// TIA Portal project "Control PLC con HMI" (V15.1)

(* hardware
DEVICE "S7-1200 station_1"  S7-1200 Station
   slot 0: "Rack_0"  S7-1200 Rack  Rack  V1.0
   slot 1: "PLC_1"  CPU 1212C AC/DC/Rly  6ES7 212-1BD30-0XB0  V2.2
DEVICE "HMI_1"  KTP400 Basic PN
   slot 0: "KTP400 Basic PN"  KTP400 Basic PN  6AV2 123-2DB03-0AX0  14.0.0.0
   slot 1: "HMI_RT_1"  KTP400 Basic PN  6AV2 123-2DB03-0AX0  14.0.0.0
   slot 5: "HMI_1.IE_CP_1"  PROFINET Interface  14.0.0.0
      slot 1: "Interfaz PROFINET_1"  PROFINET Interface
         slot 1: "Port_1"  Port
*)

// ===== PLC "PLC_1"  CPU 1212C AC/DC/Rly =====

VAR_GLOBAL   // PLC tag table "Tabla de variables estándar"
   "Q contador" AT %M0.5 : Bool;
   "CV contador" AT %MW20 : Int;
   "PV contador" AT %MW22 : Int;
   "In contador" AT %M24.1 : Bool;
   "Down contador" AT %M0.6 : Bool;
   "QD contador" AT %M1.0 : Bool;
   "Reset contador semaforo" AT %M1.1 : Bool;
   "CV contador semaforo" AT %MW30 : Int;
   "semaforo rojo" AT %M1.2 : Bool;
   "semaforo naranja" AT %M1.3 : Bool;
   "semaforo verde" AT %M1.4 : Bool;
   "Tempo" AT %M1.5 : Bool;
   "Entrada analogica 1" AT %IW66 : Int;
   "Senal escalada 1" AT %MD32 : Real;
   "Alarma up" AT %M1.6 : Bool;
   "Alarma down" AT %M1.7 : Bool;
END_VAR

VAR_GLOBAL   // PLC tag table "Entradas"
   "ARRANQUE" AT %I0.0 : Bool;
   "PARO" AT %I0.1 : Bool;
   "Senal analogica 0" AT %IW64 : Int;
END_VAR

VAR_GLOBAL   // PLC tag table "Salidas"
   "MOTOR1" AT %Q0.0 : Bool;
END_VAR

VAR_GLOBAL   // PLC tag table "Memoria"
   "Senal analogica real 0" AT %MD2 : Real;
   "Segundos" AT %MD26 : Time;
   "senal escalada" AT %MD6 : Real;
   "Senal de control" AT %M0.2 : Bool;
END_VAR

VAR_GLOBAL   // PLC tag table "HMI"
   "ARRANQUE HMI" AT %M0.0 : Bool;
   "PARO HMI" AT %M0.1 : Bool;
   "Reset contador" AT %M24.0 : Bool;
   "Q timer" AT %M0.3 : Bool;
   "Et timer" AT %MD10 : Time;
   "Pt Timer" AT %MD14 : Time;
   "in timer" AT %M18.0 : Bool;
   "Reset timer" AT %M0.4 : Bool;
   "Load contador" AT %M0.7 : Bool;
END_VAR

DATA_BLOCK "Control analogico_DB"   // DB5
{ S7_Optimized_Access := 'TRUE' }
VERSION : 0.1
// stored: InstanceOfName Control analogico
"Control analogico"
BEGIN
END_DATA_BLOCK

// folder: System blocks/Program resources

DATA_BLOCK "IEC_Timer_0_DB"   // DB1
{ S7_Optimized_Access := 'TRUE' }
AUTHOR : Simatic
FAMILY : IEC
NAME : IEC_TMR
VERSION : 1.0
// stored: InstanceOfName IEC_TIMER
"IEC_TIMER"
BEGIN
END_DATA_BLOCK

DATA_BLOCK "IEC_Counter_0_DB"   // DB2
{ S7_Optimized_Access := 'TRUE' }
AUTHOR : Simatic
FAMILY : IEC
NAME : CNTR
VERSION : 1.0
// stored: InstanceOfName IEC_COUNTER
"IEC_COUNTER"
BEGIN
END_DATA_BLOCK

DATA_BLOCK "IEC_Timer_0_DB_1"   // DB3
{ S7_Optimized_Access := 'TRUE' }
AUTHOR : Simatic
FAMILY : IEC
NAME : IEC_TMR
VERSION : 1.0
// stored: InstanceOfName IEC_TIMER
"IEC_TIMER"
BEGIN
END_DATA_BLOCK

DATA_BLOCK "IEC_Counter_0_DB_1"   // DB4
{ S7_Optimized_Access := 'TRUE' }
AUTHOR : Simatic
FAMILY : IEC
NAME : CNTR
VERSION : 1.0
// stored: InstanceOfName IEC_COUNTER
"IEC_COUNTER"
BEGIN
END_DATA_BLOCK

// folder: (top level)

FUNCTION_BLOCK "Control analogico"   // FB1, LAD
{ S7_Optimized_Access := 'TRUE' }
VERSION : 0.1
   VAR_INPUT
      "Entrada analogica" : DInt;
      Minimo : Real;
      Maximo : Real;
      "Alarm max" : Real;
      "Alarm min" : Real;
   END_VAR
   VAR_OUTPUT
      "Senal out" : Real;
      "Alarm up" : Bool;
      "Alarm down" : Bool;
   END_VAR
   VAR_TEMP
      "Sinal norm" : Real;
   END_VAR
BEGIN

REGION Network 1
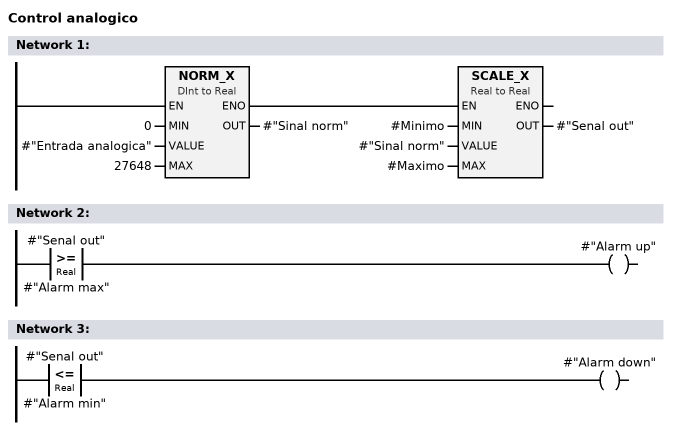
   RUNG wire#powerrail
      { S7_Templates := "[SrcType := DInt, DestType := Real]"; S7_GenerateENO := "TRUE" } Normalize(min := 0, value := #"Entrada analogica", max := 27648, out => #"Sinal norm")
      { S7_Templates := "[SrcType := Real, DestType := Real]"; S7_GenerateENO := "TRUE" } Scale(min := #Minimo, value := #"Sinal norm", max := #Maximo, out => #"Senal out")
   END_RUNG
   // the same network as SCL:
   // ENO of a box is taken as its EN; it also drops when the box reports an error
   #"Sinal norm" := NORM_X(MIN := 0, VALUE := #"Entrada analogica", MAX := 27648);
   #"Senal out" := SCALE_X(MIN := #Minimo, VALUE := #"Sinal norm", MAX := #Maximo);
END_REGION

REGION Network 2
   RUNG wire#powerrail
      { S7_Templates := "SrcType := Real" } GE_Contact(in1 := #"Senal out", in2 := #"Alarm max")
      Coil( #"Alarm up" )
   END_RUNG
   // the same network as SCL:
   #"Alarm up" := #"Senal out" >= #"Alarm max";
END_REGION

REGION Network 3
   RUNG wire#powerrail
      { S7_Templates := "SrcType := Real" } LE_Contact(in1 := #"Senal out", in2 := #"Alarm min")
      Coil( #"Alarm down" )
   END_RUNG
   // the same network as SCL:
   #"Alarm down" := #"Senal out" <= #"Alarm min";
END_REGION
END_FUNCTION_BLOCK

FUNCTION "MOTOR" : Void   // FC1, LAD
{ S7_Optimized_Access := 'TRUE' }
VERSION : 0.1
BEGIN

REGION Network 1
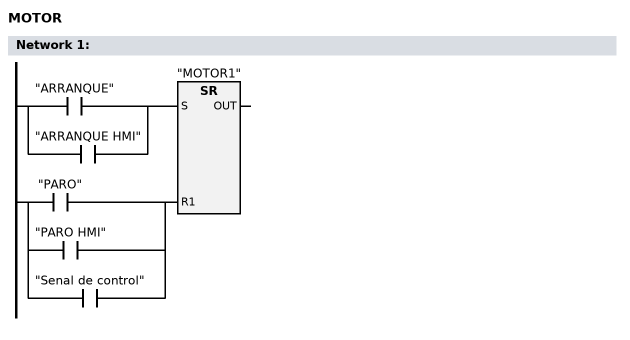
   RUNG wire#powerrail
      Contact( "ARRANQUE" )
      wire#w1
      S_SR(operand := "MOTOR1", r1 := wire#w2)
   END_RUNG
   RUNG wire#powerrail
      Contact( "ARRANQUE HMI" )
   END_RUNG wire#w1
   RUNG wire#powerrail
      Contact( "PARO" )
   END_RUNG wire#w2
   RUNG wire#powerrail
      Contact( "PARO HMI" )
   END_RUNG wire#w2
   RUNG wire#powerrail
      Contact( "Senal de control" )
   END_RUNG wire#w2
   // the same network as SCL:
   IF "ARRANQUE" OR "ARRANQUE HMI" THEN
       "MOTOR1" := TRUE;   // SR flip-flop
   END_IF;
   IF "PARO" OR "PARO HMI" OR "Senal de control" THEN "MOTOR1" := FALSE; END_IF;
END_REGION
END_FUNCTION

FUNCTION "C_ANALOGICO" : Void   // FC2, LAD
{ S7_Optimized_Access := 'TRUE' }
VERSION : 0.1
BEGIN

REGION Network 1
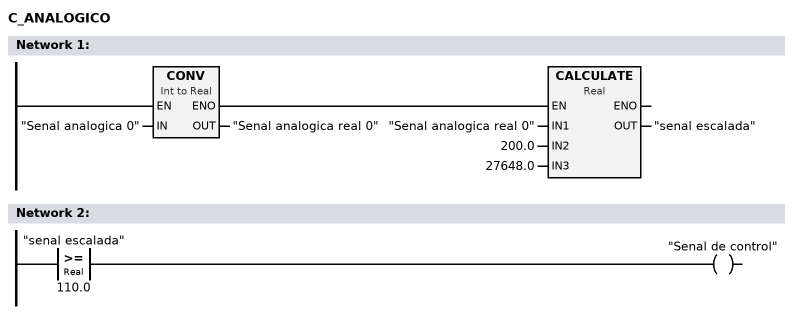
   RUNG wire#powerrail
      { S7_Templates := "[SrcType := Int, DestType := Real]"; S7_GenerateENO := "TRUE" } Convert(in := "Senal analogica 0", out => "Senal analogica real 0")
      { S7_Templates := "SrcType := Real"; S7_GenerateENO := "TRUE"; S7_Expression := "(IN1*IN2)/IN3" } Calculate(in1 := "Senal analogica real 0", in2 := 200.0, in3 := 27648.0, out => "senal escalada")
   END_RUNG
   // the same network as SCL:
   // ENO of a box is taken as its EN; it also drops when the box reports an error
   "Senal analogica real 0" := INT_TO_REAL("Senal analogica 0");
   "senal escalada" := ("Senal analogica real 0"*200.0)/27648.0;
END_REGION

REGION Network 2
   RUNG wire#powerrail
      { S7_Templates := "SrcType := Real" } GE_Contact(in1 := "senal escalada", in2 := 110.0)
      Coil( "Senal de control" )
   END_RUNG
   // the same network as SCL:
   "Senal de control" := "senal escalada" >= 110.0;
END_REGION
END_FUNCTION

FUNCTION "Temporizadores" : Void   // FC3, LAD
{ S7_Optimized_Access := 'TRUE' }
VERSION : 0.1
BEGIN

REGION Network 1
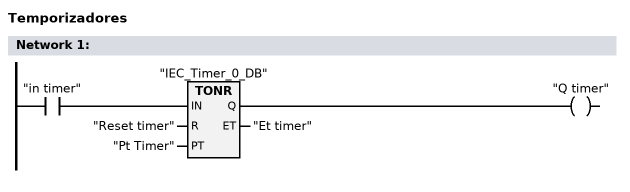
   "IEC_Timer_0_DB".TONR(IN := "in timer", R := "Reset timer", PT := "Pt Timer", ET => "Et timer");
   "Q timer" := "IEC_Timer_0_DB".Q;
END_REGION
END_FUNCTION

FUNCTION "Contador" : Void   // FC4, LAD
{ S7_Optimized_Access := 'TRUE' }
VERSION : 0.1
BEGIN

REGION Network 1
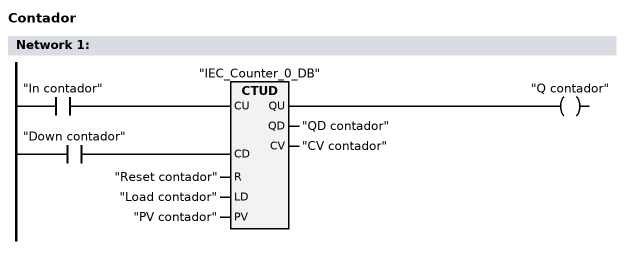
   "IEC_Counter_0_DB".CTUD(CU := "In contador",
                           CD := "Down contador",
                           R := "Reset contador",
                           LD := "Load contador",
                           PV := "PV contador",
                           QD => "QD contador",
                           CV => "CV contador");
   "Q contador" := "IEC_Counter_0_DB".QU;
END_REGION
END_FUNCTION

FUNCTION "Semaforo" : Void   // FC5, LAD
{ S7_Optimized_Access := 'TRUE' }
VERSION : 0.1
BEGIN

REGION Network 1
   // Base de tiempo
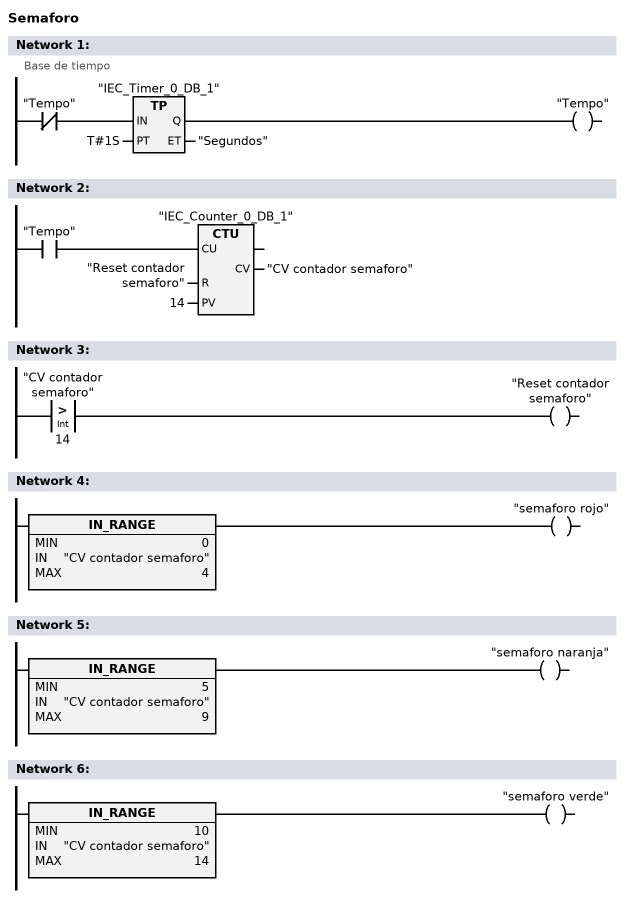
   "IEC_Timer_0_DB_1".TP(IN := NOT "Tempo", PT := T#1S, ET => "Segundos");
   "Tempo" := "IEC_Timer_0_DB_1".Q;
END_REGION

REGION Network 2
   "IEC_Counter_0_DB_1".CTU(CU := "Tempo",
                           R := "Reset contador semaforo",
                           PV := 14,
                           CV => "CV contador semaforo");
END_REGION

REGION Network 3
   RUNG wire#powerrail
      { S7_Templates := "SrcType := Int" } GT_Contact(in1 := "CV contador semaforo", in2 := 14)
      Coil( "Reset contador semaforo" )
   END_RUNG
   // the same network as SCL:
   "Reset contador semaforo" := "CV contador semaforo" > 14;
END_REGION

REGION Network 4
   RUNG wire#powerrail
      { S7_Templates := "SrcType := Int" } InRange(min := 0, in := "CV contador semaforo", max := 4)
      Coil( "semaforo rojo" )
   END_RUNG
   // the same network as SCL:
   "semaforo rojo" := (0 <= "CV contador semaforo") AND ("CV contador semaforo" <= 4);
END_REGION

REGION Network 5
   RUNG wire#powerrail
      { S7_Templates := "SrcType := Int" } InRange(min := 5, in := "CV contador semaforo", max := 9)
      Coil( "semaforo naranja" )
   END_RUNG
   // the same network as SCL:
   "semaforo naranja" := (5 <= "CV contador semaforo") AND ("CV contador semaforo" <= 9);
END_REGION

REGION Network 6
   RUNG wire#powerrail
      { S7_Templates := "SrcType := Int" } InRange(min := 10, in := "CV contador semaforo", max := 14)
      Coil( "semaforo verde" )
   END_RUNG
   // the same network as SCL:
   "semaforo verde" := (10 <= "CV contador semaforo") AND ("CV contador semaforo" <= 14);
END_REGION
END_FUNCTION

ORGANIZATION_BLOCK "Main"   // OB1, LAD, ProgramCycle
TITLE = "Main Program Sweep (Cycle)"
{ S7_Optimized_Access := 'TRUE' }
VERSION : 0.1
BEGIN

REGION Network 1
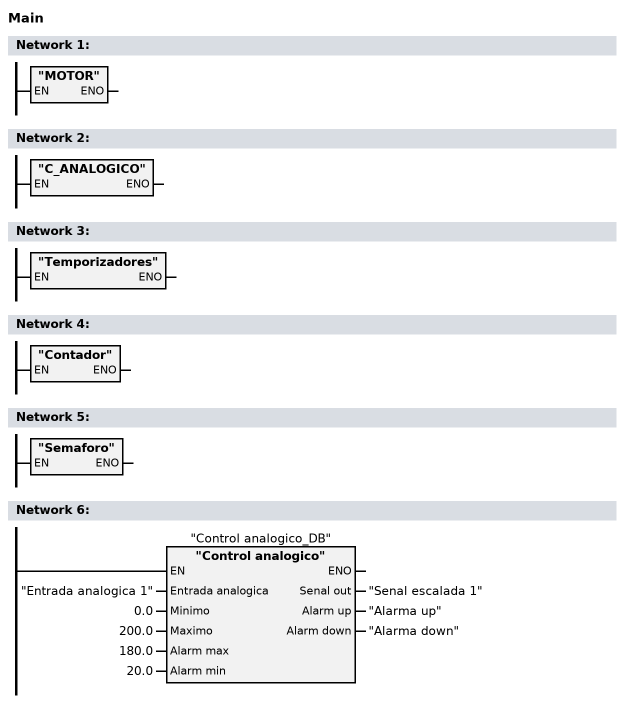
   RUNG wire#powerrail
      "MOTOR"()
   END_RUNG
   // the same network as SCL:
   "MOTOR"();
END_REGION

REGION Network 2
   RUNG wire#powerrail
      "C_ANALOGICO"()
   END_RUNG
   // the same network as SCL:
   "C_ANALOGICO"();
END_REGION

REGION Network 3
   RUNG wire#powerrail
      "Temporizadores"()
   END_RUNG
   // the same network as SCL:
   "Temporizadores"();
END_REGION

REGION Network 4
   RUNG wire#powerrail
      "Contador"()
   END_RUNG
   // the same network as SCL:
   "Contador"();
END_REGION

REGION Network 5
   RUNG wire#powerrail
      "Semaforo"()
   END_RUNG
   // the same network as SCL:
   "Semaforo"();
END_REGION

REGION Network 6
   RUNG wire#powerrail
      "Control analogico_DB"("Entrada analogica" := "Entrada analogica 1", Minimo := 0.0, Maximo := 200.0, "Alarm max" := 180.0, "Alarm min" := 20.0, "Senal out" => "Senal escalada 1", "Alarm up" => "Alarma up", "Alarm down" => "Alarma down")
   END_RUNG
   // the same network as SCL:
   "Control analogico_DB"("Entrada analogica" := "Entrada analogica 1",   // "Control analogico"
                          Minimo := 0.0,
                          Maximo := 200.0,
                          "Alarm max" := 180.0,
                          "Alarm min" := 20.0,
                          "Senal out" => "Senal escalada 1",
                          "Alarm up" => "Alarma up",
                          "Alarm down" => "Alarma down");
END_REGION
END_ORGANIZATION_BLOCK

(* ===== HMI "HMI_RT_1" =====
system functions are stored by id; their names below are inferred from use
connection "HMI_Conexión_1": ETHERNET, SMART_S7_1200_OMS

HMI tags "Tabla de variables estándar"
   "Número_imagen_variable" : UInt, internal
   "ARRANQUE HMI" : Bool = PLC "ARRANQUE HMI" AT %M0.0, 1 s
   "PARO HMI" : Bool = PLC "PARO HMI" AT %M0.1, 1 s
   "MOTOR1" : Bool = PLC MOTOR1 AT %Q0.0, 1 s
   "senal escalada" : Real = PLC "senal escalada" AT %MD6, 1 s
   "in timer" : Bool = PLC "in timer" AT %M18.0, 1 s
   "Pt Timer" : Time = PLC "Pt Timer" AT %MD14, 1 s
   "Et timer" : Time = PLC "Et timer" AT %MD10, 1 s
   "Q timer" : Bool = PLC "Q timer" AT %M0.3, 1 s
   "Reset timer" : Bool = PLC "Reset timer" AT %M0.4, 1 s
   "In contador" : Bool = PLC "In contador" AT %M24.1, 1 s
   "Q contador" : Bool = PLC "Q contador" AT %M0.5, 1 s
   "PV contador" : Int = PLC "PV contador" AT %MW22, 1 s
   "CV contador" : Int = PLC "CV contador" AT %MW20, 1 s
   "Reset contador" : Bool = PLC "Reset contador" AT %M24.0, 1 s
   "Down contador" : Bool = PLC "Down contador" AT %M0.6, 1 s
   "Load contador" : Bool = PLC "Load contador" AT %M0.7, 1 s
   "QD contador" : Bool = PLC "QD contador" AT %M1.0, 1 s
   "semaforo rojo" : Bool = PLC "semaforo rojo" AT %M1.2, 1 s
   "semaforo naranja" : Bool = PLC "semaforo naranja" AT %M1.3, 1 s
   "semaforo verde" : Bool = PLC "semaforo verde" AT %M1.4, 1 s
   "CV contador semaforo" : Int = PLC "CV contador semaforo" AT %MW30, 1 s
   "Senal escalada 1" : Real = PLC "Senal escalada 1" AT %MD32, 1 s

text list "Nombre_imagen_lista_texto": 1 'Imagen raíz'; 2 'Grafica'; 3 'Temporizadores'; 4 'Contadores'; 5 'Semaforo'

Template "Plantilla_1" 480x272
   Button "Salir" at 388,227 size 63x44; TextOff 'Salir'; PictureOff "ExitRuntime_KTP400_Basic_PN_TR"; PictureOn "ExitRuntime_KTP400_Basic_PN_TR"
      on Release: StopRuntime(0)
   Button "Template_Button" at 268,227 size 63x44; TextOff 'Text'
   Button "Template_Button_1" at 148,227 size 63x44; TextOff 'Text'
   Button "Imagen inicial" at 28,227 size 63x44; TextOff 'Imagen inicial'; PictureOff "NavigateHome_KTP400_Basic_PN_TR"; PictureOn "NavigateHome_KTP400_Basic_PN_TR"
      on Release: ActivateScreen("Pantalla principal", 0)
   SymbolicIOField "Imagen_campo_ES_simbólico" at 40,8 size 438x29; TextOff '0'; TextOn '1'; TextList "Nombre_imagen_lista_texto"
      ProcessValue <- "Número_imagen_variable"
      on Change: ActivateScreenByNumber("Número_imagen_variable", 0)

screen "Pantalla principal" 480x272, template "Plantilla_1"
   on GenerateScreen: SetTag("Número_imagen_variable", 1)
   Softkey "Softkey_F3" at 0,0 size 0x0; Authorization "Contador"
      on KeyDown: ActivateScreen("Contadores", 0)
   Softkey "Softkey_F2" at 0,0 size 0x0; Authorization "Timer"
      on KeyDown: ActivateScreen("Semaforo", 0)
   Button "Botón_1" at 36,48 size 69x25; TextOff 'I'
      on Press: function_b14e0dd5("ARRANQUE HMI", 0)
   Button "Botón_2" at 120,48 size 68x25; TextOff '0'
      on Press: function_b14e0dd5("PARO HMI", 0)
   Circle "Círculo_1" at 182,88 size 42x42
      Visibility <- "MOTOR1"
   Circle "Círculo_2" at 182,88 size 43x43
      Visibility <- "MOTOR1"
   TextField "Campo de texto_1" at 36,96 size 131x20; Text 'ESTADO DEL MOTOR'
   Bar "Barra_1" at 320,83 size 92x138; Unit °C; MinimumValue 0; MaximumValue 210
      ProcessValue <- "senal escalada"
   IOField "Campo ES_1" at 319,47 size 94x26; FormatPattern s999.9; Unit °C
      ProcessValue <- "senal escalada"
   Button "Botón_3" at 32,166 size 192x32; TextOff 'Grafica'; Authorization "Grafica"
      on Click: ActivateScreen("Grafica", 0)

screen "Grafica" 480x272
   TrendView "Visor de curvas_1" at 0,0 size 479x271
   Softkey "Softkey_F1" at 0,0 size 0x0
      on KeyDown: ActivateScreen("Pantalla principal", 0)
   Softkey "Softkey_F2" at 0,0 size 0x0
      on KeyDown: ActivateScreen("Temporizadores", 0)

screen "Temporizadores" 480x272, template "Plantilla_1"
   Softkey "Softkey_F1" at 0,0 size 0x0
      on KeyDown: ActivateScreen("Pantalla principal", 0)
   Button "Botón_1" at 30,61 size 96x32; TextOff 'IN'
      on Press: function_b14e0dd5("in timer", 0)
   Circle "Círculo_1" at 386,61 size 48x48
      Visibility <- "Q timer"
   TextField "Campo de texto_1" at 340,128 size 20x20; Text 'PT'
   IOField "Campo ES_1" at 360,124 size 96x32; FormatPattern s9999999999
      ProcessValue <- "Pt Timer"
   TextField "Campo de texto_2" at 372,73 size 14x20; Text 'Q'
   TextField "Campo de texto_3" at 340,184 size 19x20; Text 'ET'
   IOField "Campo ES_2" at 360,180 size 96x32; FormatPattern s9999999999
      ProcessValue <- "Et timer"
   Button "Botón_2" at 30,109 size 96x32; TextOff 'Reset'
      on Press: function_b14e0dd5("Reset timer", 0)
   Softkey "Softkey_F3" at 0,0 size 0x0
      on KeyDown: ActivateScreen("Contadores", 0)

screen "Contadores" 480x272, template "Plantilla_1"
   Button "Botón_1" at 41,114 size 40x32; TextOff 'In Contador'; PictureOff "Up_Arrow"
      on Press: function_b14e0dd5("In contador", 0)
   Circle "Círculo_1" at 277,66 size 48x48
      Visibility <- "QD contador"
   TextField "Campo de texto_1" at 254,83 size 23x20; Text 'QD'
   IOField "Campo ES_1" at 373,131 size 96x32; FormatPattern s99999
      ProcessValue <- "PV contador"
   TextField "Campo de texto_2" at 351,138 size 22x20; Text 'PV'
   IOField "Campo ES_2" at 373,184 size 96x32; FormatPattern s99999
      ProcessValue <- "CV contador"
   TextField "Campo de texto_3" at 351,191 size 22x20; Text 'CV'
   Button "Botón_2" at 101,111 size 114x35; TextOff 'Reset'
      on Press: function_b14e0dd5("Reset contador", 0)
   Button "Botón_3" at 41,158 size 40x32; TextOff 'In Contador'; PictureOff "Down_Arrow"
      on Press: function_b14e0dd5("Down contador", 0)
   Button "Botón_4" at 101,163 size 114x35; TextOff 'Load'
      on Press: function_b14e0dd5("Load contador", 0)
   Circle "Círculo_2" at 277,121 size 48x48
      Visibility <- "Q contador"
   TextField "Campo de texto_4" at 254,138 size 22x20; Text 'QU'
   Softkey "Softkey_F1" at 0,0 size 0x0
      on KeyDown: ActivateScreen("Pantalla principal", 0)

screen "Semaforo" 480x272, template "Plantilla_1"
   Circle "Círculo_1" at 223,34 size 48x48
      Visibility <- "semaforo rojo"
   Circle "Círculo_2" at 223,91 size 48x48
      Visibility <- "semaforo naranja"
   Circle "Círculo_3" at 223,147 size 48x48
      Visibility <- "semaforo verde"
   IOField "Campo ES_1" at 370,30 size 71x32; FormatPattern s99
      ProcessValue <- "CV contador semaforo"
   Softkey "Softkey_F1" at 0,0 size 0x0
      on KeyDown: ActivateScreen("Pantalla principal", 0)
*)